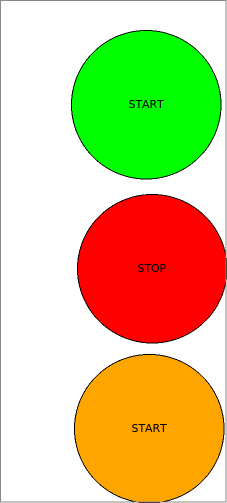
VISUALIZATION CMD  // 227x503
    Ellipse (71,30 150x149), "START"
    Ellipse (77,194 150x149), "STOP"
    Ellipse (74,354 150x149), "START"
END_VISUALIZATION

(* stored: Version 1.1.0.1, ProductVersion 3.1.4024.12
   Visu CMD: Id {514cf13c-6107-436c-b6d3-c2aa797fc2f3} *)
